FUNCTION_BLOCK BMP180 (* BMP180 I2C sensor readout *)
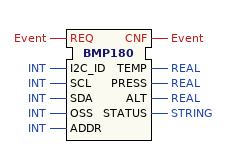
  EVENT_INPUT
    REQ; (* Request measurement *)
  END_EVENT
  EVENT_OUTPUT
    CNF; (* Measurement complete *)
  END_EVENT
  VAR_INPUT
    I2C_ID : INT; (* I2C bus id *)
    SCL : INT; (* SCL pin number *)
    SDA : INT; (* SDA pin number *)
    OSS : INT; (* Oversampling setting 0..3 *)
    ADDR : INT; (* I2C address (0x77 default) *)
  END_VAR
  VAR_OUTPUT
    TEMP : REAL; (* Temperature Celsius *)
    PRESS : REAL; (* Pressure Pa *)
    ALT : REAL; (* Altitude meters *)
    STATUS : STRING; (* Result status *)
  END_VAR
END_FUNCTION_BLOCK
